{attribute 'pack_mode=1'}
TYPE BR_SectionCommand_t :
STRUCT
    enable : BIT;
END_STRUCT
END_TYPE

(* stored: Version 1.1.0.1, ProductVersion 3.1.4024.12
   DUT BR_SectionCommand_t: Id {173215a4-f72d-491c-bb09-dc3a3ae8d538} *)
